ABB RobotStudio station: p3_1parte.rspag

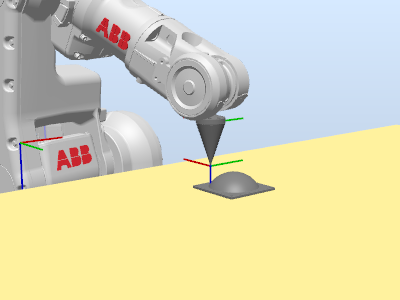
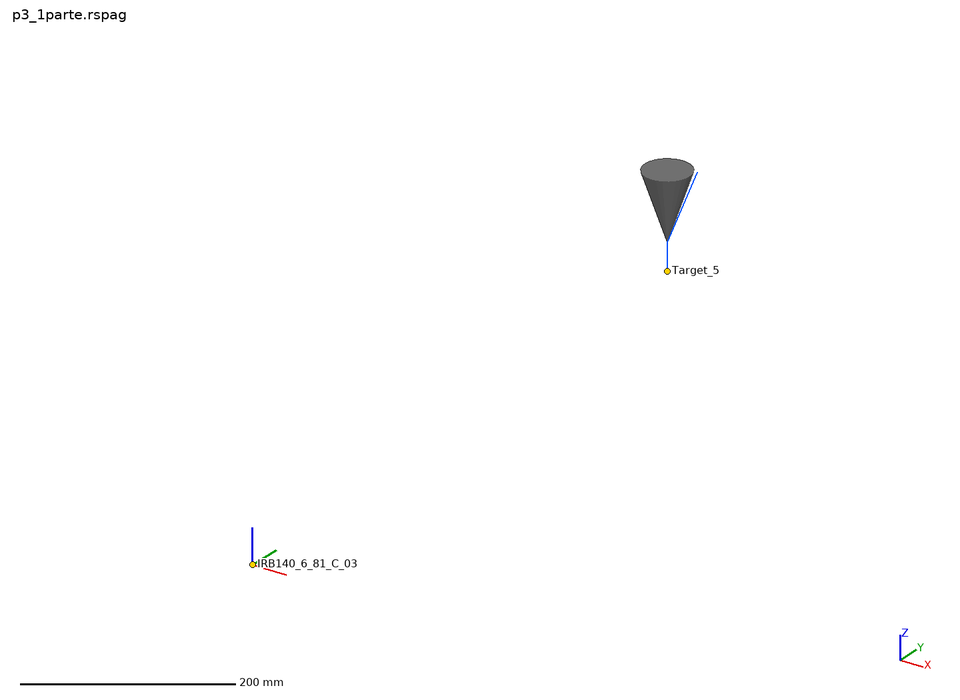
[picture v1: parts stored in the station drawn from their meshes, with robot base, taught points and paths (robot models come from the ABB library and are not in the file)]
--- station ---
Station p3_robotstudio_vacia (saved by RobotStudio 22.2.10013.1)
Controller Controlador1
  mechanical unit ROB_1: IRB140_6_81_C_03, 6 joints, base frame (0, 0, 0) mm
Layout (positions relative to the parent item):
  - printbed_hemisphere_hexagono [part, from Libraries\hemisphere.rslib] at (471.3, 85, 364.75) mm, rotated rx 90 ry 0 rz 0 deg
  - Mesa de trabajo [part, from Libraries\Mesa de trabajoDISA.rslib] at (1200, -600, -395) mm, rotated rx 0 ry 0 rz 90 deg
  - Pieza1 [part, from Libraries\Pieza_ampliacion.rslib] at (500, 0, 200) mm, rotated rx 0 ry 0 rz 90 deg
  - trazador [smart component, from Libraries\trazador.rslib] at (400, 100, 480) mm, rotated rx 180 ry 0 rz 180 deg
      connections:
        trazador.entrada_inyector -> TraceTCP.Enabled
        trazador.entrada_inyector -> ?.InputA
        ?.Output -> TraceTCP.Clear
    - TraceTCP [smart component, from Components\TraceTCP.rslib]
        properties: Robot=IRB140_6_81_C_03
  - IRB140_6_81_C_03 [mechanism, from Robots\IRB140_6_81_C_G_03.rslib] at (0, 0, 0) mm; joint values [0.245, 0.0027, 0.4523, 0, 1.1158, 0.245] (rad or m)
  - tool_laser [part] at (400, 100, 480) mm, rotated rx 180 ry 0 rz 180 deg, size 50 x 49.9 x 75 mm
  - tool_laser [mechanism] at (400, 100, 480) mm, rotated rx 180 ry 0 rz 180 deg
      TCP tool_laser at (0, 0, 75) mm
      links: Pieza_1
Attachment: trazador is attached to IRB140_6_81_C_03 / Link6
Attachment: tool_laser is attached to IRB140_6_81_C_03 / Link6
Attachment: tool_laser is attached to IRB140_6_81_C_03 / Link6
Station logic (signal -> signal, property => property):
  Controlador1.activar_mecanizado -> trazador.entrada_inyector

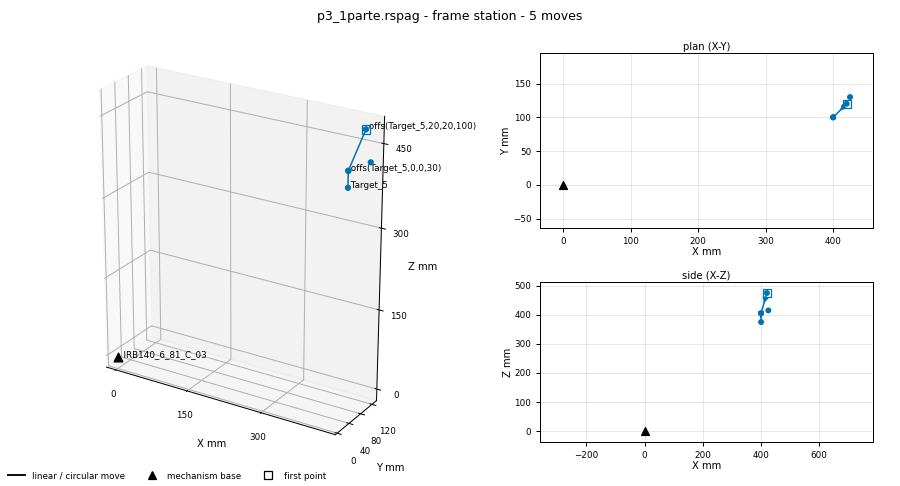
[picture p0: tool path of p3_1parte.rspag in frame station, 5 of 11 moves have a stored position in this frame; points joined in program order, loops and branches not executed]
--- Backups/Controlador1/RAPID/TASK1/PROGMOD/CalibData.mod ---
MODULE CalibData
    PERS tooldata tool_laser:=[TRUE,[[0,0,75],[1,0,0,0]],[1,[0,0,1],[1,0,0,0],0,0,0]];
    TASK PERS wobjdata Workobject:=[FALSE,TRUE,"",[[0,0,0],[1,0,0,0]],[[286.627001811,-193.490730871,464.561998296],[0.002682563,0.707605914,0.706600086,0.001729967]]];
ENDMODULE

--- Backups/Controlador1/RAPID/TASK1/PROGMOD/MainModule.mod ---
        MODULE MainModule
    	CONST robtarget Target_5:= [[400,100,375],[0,0,1,0],[0,0,0,0],[9E9,9E9,9E9,9E9,9E9,9E9]];
	    VAR socketdev socket_server;
	    VAR socketdev socket_client;
	    VAR string cadena_datos_recibida := "";
    	VAR string cadena_ACK := "ok";
	    VAR string client_ip := "";
	    VAR string server_ip := "158.42.206.38";
	    VAR num puerto := 11000;
	    VAR num valor := 0;
	    VAR bool errordato := FALSE;
    	VAR bool continuar:=TRUE;
	    VAR num desplazax:=0;
	    VAR num desplazay:=0;
	    VAR num desplazaz:=0;

	    VAR string string_x:="";
	    VAR string string_y:="";
	    VAR string string_z:="";

    	VAR num tipo_movimiento;
    	VAR num coorX;
    	VAR num coorY;
    	VAR num coorZ;
    	VAR num q1;
    	VAR num q2;
    	VAR num q3;
    	VAR num q4;

    	VAR num longitud_trama;
    	VAR bool ok;
    	VAR num pos_campo1;
    	VAR num pos_campo2;
    	VAR num pos_campo3;
    	VAR num pos_campo4;
    	VAR num pos_campo5;
   	    VAR num pos_campo6;
    	VAR num pos_campo7;
    	VAR num pos_campo8;
    	VAR string cadena1;
    	VAR string cadena2;
    	VAR string cadena3;
    	VAR string cadena4;
    	VAR string cadena5;
    	VAR string cadena6;
    	VAR string cadena7;
    	VAR string cadena8;

    	VAR robtarget posicion_robot;
        VAR bool first;

    	PROC lectura_sockets()
           SocketReceive socket_client\Str:=cadena_datos_recibida;
           !TPWrite cadena_datos_recibida;

           !Calcular longitud de la cadena
           longitud_trama:=StrLen(cadena_datos_recibida);

           !Lectura de la string
           IF longitud_trama>0 THEN
                    pos_campo1:=StrFind(cadena_datos_recibida,1,";");
                    pos_campo2:=StrFind(cadena_datos_recibida,pos_campo1+1,";");
                    pos_campo3:=StrFind(cadena_datos_recibida,pos_campo2+1,";");
                    pos_campo4:=StrFind(cadena_datos_recibida,pos_campo3+1,";");
                    pos_campo5:=StrFind(cadena_datos_recibida,pos_campo4+1,";");
                    pos_campo6:=StrFind(cadena_datos_recibida,pos_campo5+1,";");
                    pos_campo7:=StrFind(cadena_datos_recibida,pos_campo6+1,";");
                    pos_campo8:=StrFind(cadena_datos_recibida,pos_campo7+1,";");

                    cadena1:=StrPart(cadena_datos_recibida,1,pos_campo1-1);
                    cadena2:=StrPart(cadena_datos_recibida,pos_campo1+1,pos_campo2-pos_campo1-1);
                    cadena3:=StrPart(cadena_datos_recibida,pos_campo2+1,pos_campo3-pos_campo2-1);
                    cadena4:=StrPart(cadena_datos_recibida,pos_campo3+1,pos_campo4-pos_campo3-1);
                    cadena5:=StrPart(cadena_datos_recibida,pos_campo4+1,pos_campo5-pos_campo4-1);
                    cadena6:=StrPart(cadena_datos_recibida,pos_campo5+1,pos_campo6-pos_campo5-1);
                    cadena7:=StrPart(cadena_datos_recibida,pos_campo6+1,pos_campo7-pos_campo6-1);
                    cadena8:=StrPart(cadena_datos_recibida,pos_campo7+1,pos_campo8-pos_campo7-1);

                    ok:=StrToVal(cadena1,tipo_movimiento);
                    ok:=StrToVal(cadena2,coorX);
                    ok:=StrToVal(cadena3,coorY);
                    ok:=StrToVal(cadena4,coorZ);
                    ok:=StrToVal(cadena5,q1);
                    ok:=StrToVal(cadena6,q2);
                    ok:=StrToVal(cadena7,q3);
                    ok:=StrToVal(cadena8,q4);
                ELSE
                	TPWrite "error en recepci n trama";
            	endif
    	ENDPROC


    	PROC inicializa_sockets()
        	SocketCreate socket_server;
		    SocketBind socket_server, server_ip, puerto;
		    SocketListen socket_server;
		    SocketAccept socket_server, socket_client\ClientAddress:=client_ip;
    	ENDPROC


	PROC main()
        	inicializa_sockets;
            Reset activar_mecanizado;
            TPWrite "Connecion establecida";

        	MoveJ offs(Target_5, 20, 20,100),v100,fine,tool_laser\WObj:=wobj0;
            MoveL offs(Target_5, 0, 0,30),v10,fine,tool_laser\WObj:=wobj0;
            MoveL Target_5,v5,fine,tool_laser\WObj:=wobj0;
        	continuar:=TRUE;
            first:=TRUE;

	       WHILE continuar DO
                  lectura_sockets;
                  TPWrite "tipo_movimiento: "\Num:= tipo_movimiento;
                  TPWrite "coorX: "\Num:= coorX;
                  TPWrite "coorY: "\Num:= coorY;
                  TPWrite "coorZ: "\Num:= coorZ;
                  TPWrite "q1: "\Num:= q1;
                  TPWrite "q2: "\Num:= q2;
                  TPWrite "q3: "\Num:= q3;
                  TPWrite "q4: "\Num:= q4;
                  posicion_robot:=CRobT();
                  posicion_robot := Offs(Target_5,coorX,coorY,coorZ);
                  posicion_robot.rot := [q1,q2,q3,q4];
                  TEST tipo_movimiento
                      CASE 0:
                        Reset activar_mecanizado;
                        IF first THEN
                            MoveJ Offs(posicion_robot,0,0,8),v100,fine,tool_laser\WObj:=wobj0;
                            MoveJ posicion_robot,v100,fine,tool_laser\WObj:=wobj0;
                            first := FALSE;
                        ELSE
                            MoveJ Offs(CRobT(),0,0,15), v100, fine, tool_laser\WObj:=wobj0;
                            MoveJ Offs(Target_5,25,30,40), v100, fine, tool_laser\WObj:=wobj0;
                            MoveJ Offs(posicion_robot,0,0,25),v100,fine,tool_laser\WObj:=wobj0;
                            MoveJ posicion_robot,v100,fine,tool_laser\WObj:=wobj0;
                        ENDIF
                      CASE 1:
                        Set activar_mecanizado;
                        MoveL posicion_robot,v50,fine,tool_laser\WObj:=wobj0;
                      CASE 2:
                        continuar := False;
                  ENDTEST

                  SocketSend socket_client\Str:=cadena_ACK;

	      ENDWHILE

          MoveJ offs(Target_5,0,0,30),v100,fine,tool_laser\WObj:=wobj0;
	      SocketClose socket_server;
          TPWrite "Fin de mecanizado";
	ENDPROC
    PROC Path_10()

    ENDPROC
ENDMODULE

--- Backups/Controlador1/SYSPAR/EIO.cfg ---
EIO:CFG_1.0:6:1::
#
EIO_SIGNAL:

      -Name "activar_mecanizado" -SignalType "DO" -Access "All"
